INTERFACE I_Request EXTENDS I_Disposable

PROPERTY PUBLIC CreatedTimestamp : I_Timestamp
GET
END_GET
END_PROPERTY

PROPERTY PUBLIC Header : I_Header
GET
END_GET
END_PROPERTY

PROPERTY PUBLIC PayloadAddress : POINTER TO STRING
GET
END_GET
END_PROPERTY

PROPERTY PUBLIC PayloadSizeInBytes : UDINT
GET
END_GET
END_PROPERTY

END_INTERFACE

(* stored: Version 1.1.0.1, ProductVersion 3.1.4024.12
   Itf I_Request: Id {09fb0484-0921-4add-a143-8e5b5a4ec79b}
   Property CreatedTimestamp: Id {6654dbac-bbdc-4e29-abd7-f7bae031a16b}
   Get Get: Id {a8827976-4218-49a8-958a-254625df3344}
   Property Header: Id {e48d46f2-b1ae-4764-81c7-c961d7cf6a85}
   Get Get: Id {aa2814e0-af57-4ffe-a8c4-7e1da4004afd}
   Property PayloadAddress: Id {f0a14312-a7f3-4fde-a466-6fa0210857d4}
   Get Get: Id {9d2ca32a-6748-482e-86dd-a46e8d522a62}
   Property PayloadSizeInBytes: Id {9682ec78-1d85-4cc2-95d0-414b63bd0d84}
   Get Get: Id {d4101461-c609-41eb-b582-700fc702336c} *)
